FUNCTION FUN_GetLowByte : BYTE
VAR_INPUT
	wIn			:WORD;			
END_VAR
VAR
	byLow		:BYTE;
END_VAR


// Get the high byte value from the word
byLow.0 := wIn.0;
byLow.1 := wIn.1;
byLow.2 := wIn.2;
byLow.3 := wIn.3;
byLow.4 := wIn.4;
byLow.5 := wIn.5;
byLow.6 := wIn.6;
byLow.7 := wIn.7;

// Return value
FUN_GetLowByte := byLow;

END_FUNCTION

(* stored: Version 1.1.0.1, ProductVersion 3.1.4024.12
   POU FUN_GetLowByte: Id {f1c1033d-197c-472d-831b-7045c44ff0bf}, SpecialFunc None *)
